FUNCTION_BLOCK Sensor (* Template for an empty basic function block *)
  (* Standard: 61499-2 *)
  (* Version 1.0, 2019-03-19, Duc Do Tran, OFFIS e.V. *)
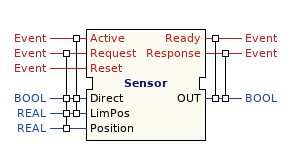
  EVENT_INPUT
    Active WITH Direct, LimPos;
    Request WITH Direct, LimPos, Position;
    Reset;
  END_EVENT
  EVENT_OUTPUT
    Ready WITH OUT;
    Response WITH OUT;
  END_EVENT
  VAR_INPUT
    Direct : BOOL;
    LimPos : REAL := 180;
    Position : REAL;
  END_VAR
  VAR_OUTPUT
    OUT : BOOL := FALSE;
  END_VAR
  VAR
    trigger : BOOL; (* Internal Variable *)
    i : USINT := 0; (* Internal Variable *)
    change : BOOL; (* Internal Variable *)
  END_VAR
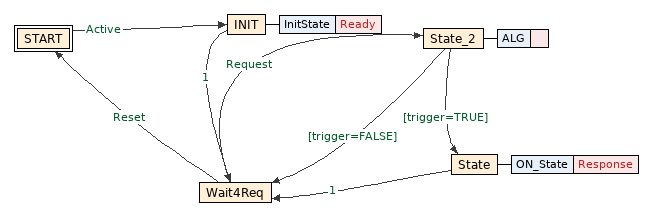
  EC_STATES
    START; (* Initial State *)
    State : ON_State -> Response;
    State_2 : ALG;
    INIT : InitState -> Ready;
    Wait4Req;
  END_STATES
  EC_TRANSITIONS
    State_2 TO Wait4Req := [trigger=FALSE];
    State_2 TO State := [trigger=TRUE];
    START TO INIT := Active;
    Wait4Req TO State_2 := Request;
    State TO Wait4Req := 1;
    Wait4Req TO START := Reset;
    INIT TO Wait4Req := 1;
  END_TRANSITIONS
  ALGORITHM ON_State IN ST: (* new algorithm *)
OUT := TRUE;
trigger := FALSE;
  END_ALGORITHM
  ALGORITHM ALG IN ST: (* new algorithm *)
IF (Direct = FALSE) THEN //Run to LS2
	IF (Position >= LimPos) THEN
		IF (change = FALSE) THEN
			change := TRUE;
			trigger := TRUE;
		END_IF;
	ELSE
		IF (change = TRUE) THEN
			change := FALSE;
			OUT := FALSE;
		END_IF;
		trigger := FALSE;
	END_IF;
ELSE
	IF (Position <= LimPos) THEN
		IF (change = FALSE) THEN
			change := TRUE;
			trigger := TRUE;
		END_IF;
	ELSE
		IF (change = TRUE) THEN
			change := FALSE;
			OUT := FALSE;
		END_IF;
		trigger := FALSE;
	END_IF;
END_IF;
  END_ALGORITHM
  ALGORITHM InitState IN ST: (* new algorithm *)
/*IF (Direct = TRUE) THEN
	OUT := FALSE;
ELSE
	OUT :=TRUE;
END_IF;*/
OUT := FALSE;
trigger := FALSE;
change := FALSE;
  END_ALGORITHM
END_FUNCTION_BLOCK
